TYPE TcaSegmentDoorStatus :
STRUCT
    ActionDescription : STRING(100);	         
	Safe : BOOL;
	Open : BOOL;
	
END_STRUCT
END_TYPE

(* stored: Version 1.1.0.1
   DUT TcaSegmentDoorStatus: Id {dcb1980d-226d-41a5-9da5-5874f243800d} *)
